(* CODESYS project tcdevicebase.library
   Company: TcNexa
   DefaultNamespace: TcNexa_Devices_Base_TcDeviceBase
   Version: 1.0.0.0
   Placeholder: TcDeviceBase
   Author: ATI Software Engineering
   Title: TcDeviceBase

Project tree, tasks and I/O mapping:
  libraries: Tc2_Standard, * (Beckhoff Automation GmbH); Tc2_System, * (Beckhoff Automation GmbH); Tc3_Module, * (Beckhoff Automation GmbH); TcProcess, * (TcNexa)
  Base/
    DUTs/
      data type ST_MethodState
    POUs/
      function block FB_DeviceBase [ST]: _appendErrorDescription, _getBusyDescription, _getErrorDescription, _getErrorIdDescription, _getStepMissingError, _getTimeoutDescription, _getWarningIdDescription, _methodFooter, _methodHeader, FB_init, FB_main
  GVLs/
    global variables GVL_DeviceBase
  POUs/
    program PRG_TEST [ST]
  Version/
    global variables Global_Version
*)

// Base/DUTs/ST_MethodState
TYPE ST_MethodState :
STRUCT
	init		: BOOL;
	execute		: BOOL;
	timeout		: BOOL;
END_STRUCT
END_TYPE

// GVLs/GVL_DeviceBase
VAR_GLOBAL
	DEFAULT_DEVICE_TIMEOUT			: TIME:= Tc2_System.DEFAULT_ADS_TIMEOUT;
	ERROR_DESCRIPTION_DELIMITER		: STRING:= '$L -> ';
END_VAR

// Version/Global_Version
{attribute 'TcGenerated'}
{attribute 'no-analysis'}
{attribute 'linkalways'}
// This function has been automatically generated from the project information.
VAR_GLOBAL CONSTANT
	{attribute 'const_non_replaced'}
	stLibVersion_TcDeviceBase : ST_LibVersion := (iMajor := 1, iMinor := 0, iBuild := 0, iRevision := 0, nFlags := 0, sVersion := '1.0.0.0');
END_VAR

// Base/POUs/FB_DeviceBase
FUNCTION_BLOCK ABSTRACT FB_DeviceBase
VAR
	_Step					: TcNexa_Components_TcProcess.FB_ProcessStep;
	_InternalResponse		: TcNexa_Components_TcProcess.FB_MethodResponse;
	_calledMethod			: STRING;
	_tmpText				: Tc2_System.T_MaxString;
	_methodTimeout			: Tc2_Standard.TON;
	_methodState			: ST_MethodState;
	_methodName				: STRING;
	_executeMethod			: BOOL;
	_cellTag				: STRING;
	_stationTag				: STRING;
	_name					: STRING;
	_tag					: STRING;
	_nameTag				: STRING;
	_methodTime				: TIME:= Tc2_System.DEFAULT_ADS_TIMEOUT;
	_noMethodCalledTrigger	: Tc2_Standard.R_TRIG;
END_VAR

METHOD PROTECTED _appendErrorDescription : Tc2_System.T_MaxString
VAR_INPUT
	description		: Tc2_System.T_MaxString;
END_VAR
_appendErrorDescription:= Tc2_Standard.CONCAT(STR1:= _nameTag, STR2:= ' ');
_appendErrorDescription:= Tc2_Standard.CONCAT(STR1:= _appendErrorDescription, STR2:= _methodName);
_appendErrorDescription:= Tc2_Standard.CONCAT(STR1:= _appendErrorDescription, STR2:= ' error');
_appendErrorDescription:= Tc2_Standard.CONCAT(STR1:= _appendErrorDescription, STR2:= ERROR_DESCRIPTION_DELIMITER);
_appendErrorDescription:= Tc2_Standard.CONCAT(STR1:= _appendErrorDescription, STR2:= description);
END_METHOD

METHOD PROTECTED _getBusyDescription : Tc2_System.T_MaxString
VAR_INPUT
	description		: Tc2_System.T_MaxString;
END_VAR
_getBusyDescription:= Tc2_Standard.CONCAT(STR1:= _nameTag, STR2:= ' ');
_getBusyDescription:= Tc2_Standard.CONCAT(STR1:= _getBusyDescription, STR2:= _methodName);
_getBusyDescription:= Tc2_Standard.CONCAT(STR1:= _getBusyDescription, STR2:= ' ');
_getBusyDescription:= Tc2_Standard.CONCAT(STR1:= _getBusyDescription, STR2:= description);
END_METHOD

METHOD PROTECTED _getErrorDescription : Tc2_System.T_MaxString
VAR_INPUT
	error		: STRING;
END_VAR
_getErrorDescription:= _nameTag;
IF (_methodName <> '') THEN
	_getErrorDescription:= Tc2_Standard.CONCAT(STR1:= _getErrorDescription, STR2:= ' ');
	_getErrorDescription:= Tc2_Standard.CONCAT(STR1:= _getErrorDescription, STR2:= _methodName);
END_IF
_getErrorDescription:= Tc2_Standard.CONCAT(STR1:= _getErrorDescription, STR2:= ' error ');
_getErrorDescription:= Tc2_Standard.CONCAT(STR1:= _getErrorDescription, STR2:= error);
END_METHOD

METHOD PROTECTED _getErrorIdDescription : Tc2_System.T_MaxString
VAR_INPUT
	errorId		: UDINT;
END_VAR
_getErrorIdDescription:= Tc2_Standard.CONCAT(STR1:= _nameTag, STR2:= ' ');
_getErrorIdDescription:= Tc2_Standard.CONCAT(STR1:= _getErrorIdDescription, STR2:= _methodName);
_getErrorIdDescription:= Tc2_Standard.CONCAT(STR1:= _getErrorIdDescription, STR2:= ' error with errorId ');
_getErrorIdDescription:= Tc2_Standard.CONCAT(STR1:= _getErrorIdDescription, STR2:= UDINT_TO_STRING(errorId));
_getErrorIdDescription:= Tc2_Standard.CONCAT(STR1:= _getErrorIdDescription, STR2:= '');
END_METHOD

METHOD PROTECTED _getStepMissingError : Tc2_System.T_MaxString
VAR_INPUT
END_VAR
VAR
END_VAR
_getStepMissingError:= Tc2_Standard.CONCAT(STR1:= _nameTag, STR2:= ' ');
_getStepMissingError:= Tc2_Standard.CONCAT(STR1:= _getStepMissingError, STR2:= _methodName);
_getStepMissingError:= Tc2_Standard.CONCAT(STR1:= _getStepMissingError, STR2:= ' error step ');	
_getStepMissingError:= Tc2_Standard.CONCAT(STR1:= _getStepMissingError, STR2:= INT_TO_STRING(_Step.actual));	
_getStepMissingError:= Tc2_Standard.CONCAT(STR1:= _getStepMissingError, STR2:= ' not found');
END_METHOD

METHOD PROTECTED _getTimeoutDescription : Tc2_System.T_MaxString
VAR_INPUT
END_VAR
_getTimeoutDescription:= Tc2_Standard.CONCAT(STR1:= _name, STR2:= ' timeout during ');
_getTimeoutDescription:= Tc2_Standard.CONCAT(STR1:= _getTimeoutDescription, STR2:= _methodName);
END_METHOD

METHOD PROTECTED _getWarningIdDescription : Tc2_System.T_MaxString
VAR_INPUT
	Id		: UDINT;
END_VAR
_getWarningIdDescription:= Tc2_Standard.CONCAT(STR1:= _nameTag, STR2:= ' ');
_getWarningIdDescription:= Tc2_Standard.CONCAT(STR1:= _getWarningIdDescription, STR2:= _methodName);
_getWarningIdDescription:= Tc2_Standard.CONCAT(STR1:= _getWarningIdDescription, STR2:= ' warning with warningId ');
_getWarningIdDescription:= Tc2_Standard.CONCAT(STR1:= _getWarningIdDescription, STR2:= UDINT_TO_STRING(Id));
_getWarningIdDescription:= Tc2_Standard.CONCAT(STR1:= _getWarningIdDescription, STR2:= '');
END_METHOD

METHOD PROTECTED _methodFooter
VAR_INPUT
	Response		: REFERENCE TO TcNexa_Components_TcProcess.FB_MethodResponse;
END_VAR
IF NOT _InternalResponse.busy THEN _calledMethod:= ''; END_IF
IF __ISVALIDREF(Response) THEN Response.copyFrom(Response:= _InternalResponse); END_IF
END_METHOD

METHOD PROTECTED _methodHeader : ST_MethodState
VAR_INPUT
	methodName		: Tc2_System.T_MaxString;
END_VAR
_methodName:= methodName;

IF (_calledMethod = '') THEN
	_calledMethod:= methodName;
	_Step.init();
	_methodTimeout(IN:= FALSE);
	_methodHeader.init:= TRUE;
	_methodHeader.execute:= TRUE;
	_executeMethod:= TRUE;
	_InternalResponse.setBusy(description:= methodName);
ELSIF (_calledMethod = methodName) THEN
	_executeMethod:= TRUE;
	_methodTimeout(IN:= TRUE, PT:= _methodTime);
	IF _methodTimeout.Q THEN
		_InternalResponse.setFail(description:= _getTimeoutDescription());
		_methodHeader.timeout:= TRUE;
	ELSE
		_tmpText:= _getBusyDescription(description:= 'in progress...');
		_InternalResponse.setBusy(description:= _tmpText);
		_methodHeader.execute:= TRUE;
	END_IF
ELSE
	_tmpText:= _getBusyDescription(description:= 'in progress...');
	_InternalResponse.setBusy(description:= _tmpText);
END_IF
END_METHOD

METHOD FB_init : BOOL
VAR_INPUT
	bInitRetains 	: BOOL; // if TRUE, the retain variables are initialized (warm start / cold start)
	bInCopyCode 	: BOOL;  // if TRUE, the instance afterwards gets moved into the copy code (online change)
	cellTag			: STRING;
	stationTag		: STRING;
	name			: STRING;
	tag				: STRING;
	timeout			: TIME;
END_VAR
THIS^._cellTag:= cellTag;
THIS^._stationTag:= stationTag;
THIS^._name:= name;
THIS^._tag:= tag;
THIS^._methodTime:= timeout;

_nameTag:= name;
IF (tag <> '') THEN
	IF (name <> '') THEN
		_nameTag:= Tc2_Standard.CONCAT(STR1:= _nameTag, STR2:= ' ');
	END_IF
	_nameTag:= Tc2_Standard.CONCAT(STR1:= _nameTag, STR2:= '(');
	_nameTag:= Tc2_Standard.CONCAT(STR1:= _nameTag, STR2:= tag);
	_nameTag:= Tc2_Standard.CONCAT(STR1:= _nameTag, STR2:= ')');
END_IF
END_METHOD

METHOD PUBLIC FB_main
VAR_INPUT
END_VAR
_noMethodCalledTrigger(CLK:= (_calledMethod = ''));

IF (_calledMethod <> '') AND NOT _executeMethod THEN
	_calledMethod:= '';
END_IF

_executeMethod:= FALSE;
END_METHOD

END_FUNCTION_BLOCK

// POUs/PRG_TEST
PROGRAM PRG_TEST
VAR
//	_test			: FB_DeviceBase;
END_VAR

END_PROGRAM
